TYPE ST_Point :
STRUCT
x:REAL;
y:REAL;
z:REAL;
END_STRUCT
END_TYPE

(* stored: Version 1.1.0.1, ProductVersion 3.1.4024.12
   DUT ST_Point: Id {b2c3d4e5-f6a7-4b8c-9d0e-1f2a3b4c5d6e} *)
